INTERFACE IUnsupportedEventHandler EXTENDS IEventHandlerBase

END_INTERFACE

(* stored: Version 1.1.0.1, ProductVersion 3.1.4024.4
   Itf IUnsupportedEventHandler: Id {3def3755-5dd4-4134-83ba-9efa7b99ab72} *)
